{attribute addProperty BoxType "EJ2522-0000-0022"}
{attribute addProperty Id "Target_counter_valueAT %Q*UDINT324"}
{attribute addProperty CRC "960858524"}
{attribute addProperty SizeInBites "32"}
{attribute addProperty SizeInBytes "4"}
TYPE PTO_Target_Channel_3945899C :
STRUCT
	{attribute addProperty Name "Target_counter_value"}
	Target_counter_value AT %Q* : UDINT;
END_STRUCT
END_TYPE

(* stored: Version 1.2.0.0, ProductVersion 3.1.4024.9
   DUT PTO_Target_Channel_3945899C: Id {94ce43f9-1620-4924-a504-9f0d25245720} *)
